INTERFACE ITF_GroupElement1 EXTENDS ITF_BaseGroupElement

END_INTERFACE

(* stored: Version 1.1.0.1, ProductVersion 3.1.4024.15
   Itf ITF_GroupElement1: Id {c6455967-957f-40c7-9f4a-93369d417bd9} *)
